% RSLogix 500 project CROWN_CITRUS_BIN_WASH_FROM_USB_AUG_30_2021_BAK438.RSS, saved by version 11.00.00.00 %
PROJECT "JBT BIN"    % processor: MicroLogix 1400 %

PROGRAM FILES
  LAD 2 "MAIN"  9 rungs
  LAD 3 "START_UP"  4 rungs
  LAD 4 "ENCODER"  6 rungs
  LAD 5 "CRADLE"  25 rungs
  LAD 6 "BRUSH"  7 rungs
  LAD 7 "TANK"  18 rungs
  LAD 8 "AUXILARY"  4 rungs
  LAD 9 "FAULTS"  29 rungs
  LAD 10 "HSC"  2 rungs

DATA FILES
  O0 OUTPUT  6 elements
  I1 INPUT  8 elements
  S2 STATUS  66 elements
  B3 BINARY  4 elements
  T4 TIMER  19 elements
  C5 COUNTER  1 elements
  R6 CONTROL  1 elements
  N7 INTEGER  7 elements
  F8 FLOAT  1 elements
  L9   3 elements
  L10   2 elements

LADDER 2 "MAIN"
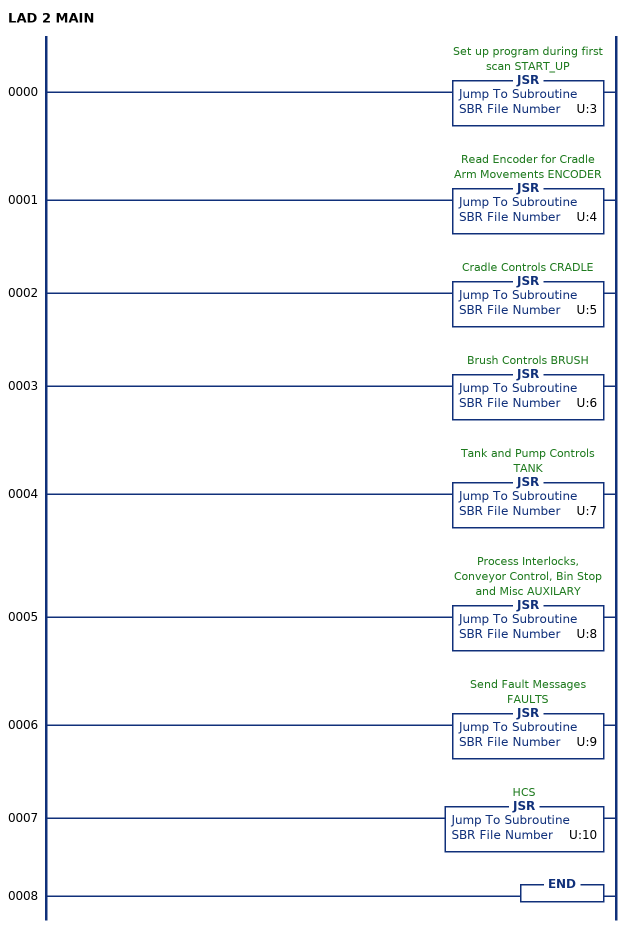
% Rung: 0 %
SOR JSR U:3 EOR
%   U:3  START_UP  "Set up program during first scan" %
% Rung: 1 %
SOR JSR U:4 EOR
%   U:4  ENCODER  "Read Encoder for Cradle Arm Movements" %
% Rung: 2 %
SOR JSR U:5 EOR
%   U:5  CRADLE  "Cradle Controls" %
% Rung: 3 %
SOR JSR U:6 EOR
%   U:6  BRUSH  "Brush Controls" %
% Rung: 4 %
SOR JSR U:7 EOR
%   U:7  TANK  "Tank and Pump Controls" %
% Rung: 5 %
SOR JSR U:8 EOR
%   U:8  AUXILARY  "Process Interlocks, Conveyor Control, Bin Stop and Misc" %
% Rung: 6 %
SOR JSR U:9 EOR
%   U:9  FAULTS  "Send Fault Messages" %
% Rung: 7 %
SOR JSR U:10 EOR
%   U:10  HCS %
% Rung: 8 %
SOR END EOR

LADDER 3 "START_UP"
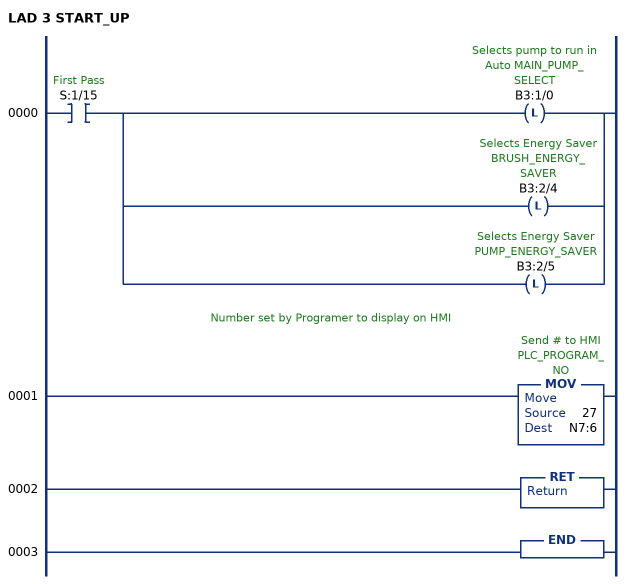
% Rung: 0 %
SOR XIC S:1/15 BST OTL B3:1/0 NXB BST OTL B3:2/4 NXB OTL B3:2/5 BND BND EOR
%   S:1/15  "First Pass" %
%   B3:1/0  MAIN_PUMP_SELECT  "Selects pump to run in Auto" %
%   B3:2/4  BRUSH_ENERGY_SAVER  "Selects Energy Saver" %
%   B3:2/5  PUMP_ENERGY_SAVER  "Selects Energy Saver" %
% Rung: 1 %
% Number set by Programer to display on HMI %
SOR MOV 27 N7:6 EOR
%   N7:6  PLC_PROGRAM_NO  "Send # to HMI" %
% Rung: 2 %
SOR RET EOR
% Rung: 3 %
SOR END EOR

LADDER 4 "ENCODER"
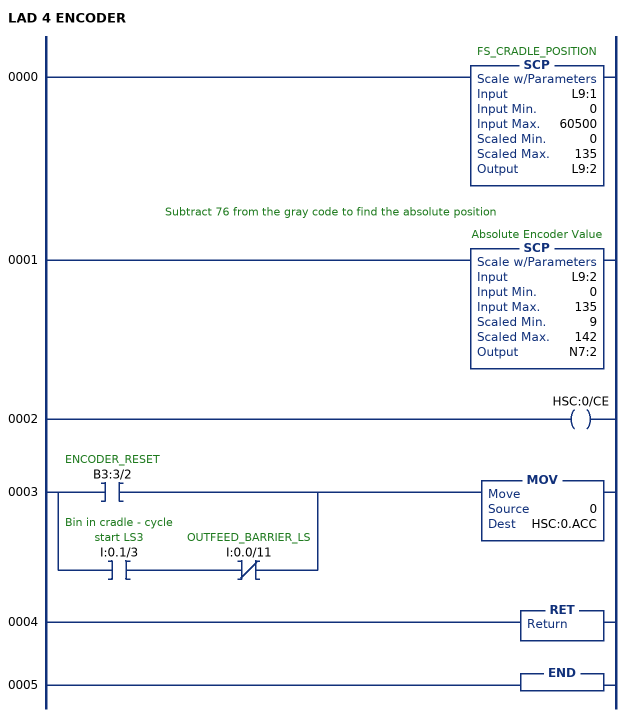
% Rung: 0 %
SOR SCP L9:1 0 60500 0 135 L9:2 EOR
%   L9:1  HSC_RAW_ACC %
%   L9:2  FS_CRADLE_POSITION %
% Rung: 1 %
% Subtract 76 from the gray code to find the absolute position %
SOR SCP L9:2 0 135 9 142 N7:2 EOR
%   L9:2  FS_CRADLE_POSITION %
%   N7:2  "Absolute Encoder Value" %
% Rung: 2 %
SOR OTE HSC:0/CE EOR
% Rung: 3 %
SOR BST XIC B3:3/2 NXB XIC I:0.1/3 XIO I:0.0/11 BND MOV 0 HSC:0.ACC EOR
%   B3:3/2  ENCODER_RESET %
%   I:0.1/3  LS3  "Bin in cradle - cycle start" %
%   I:0.0/11  OUTFEED_BARRIER_LS %
% Rung: 4 %
SOR RET EOR
% Rung: 5 %
SOR END EOR

LADDER 5 "CRADLE"
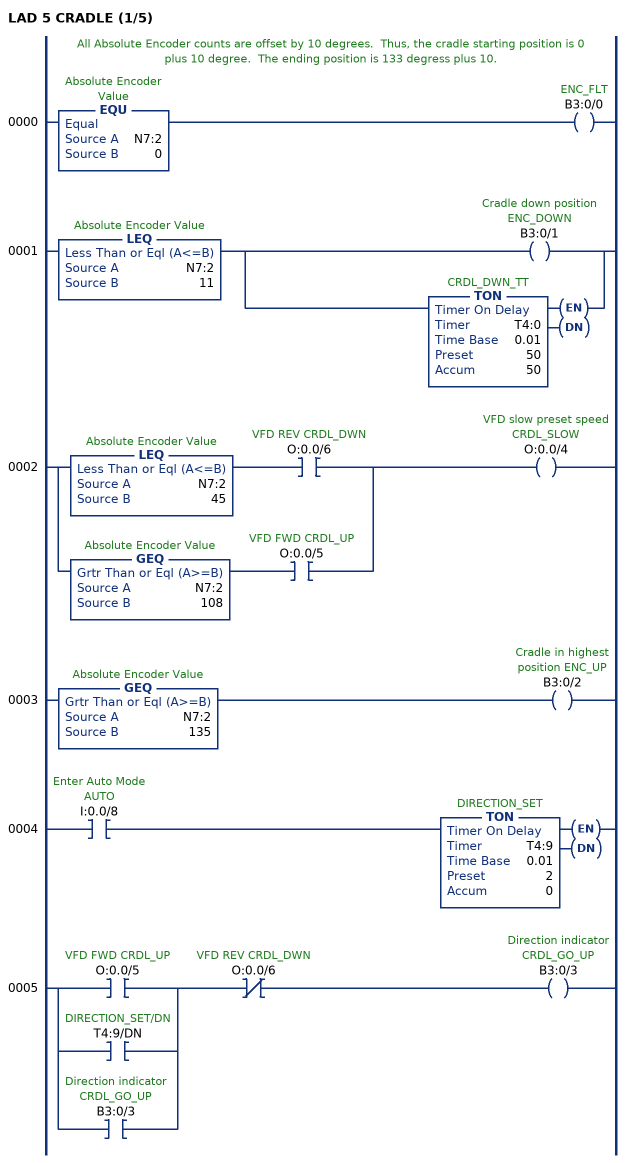
% Rung: 0 %
% All Absolute Encoder counts are offset by 10 degrees.  Thus, the cradle starting position is 0 plus 10 degree.  The ending position is 133 degress plus 10. %
SOR EQU N7:2 0 OTE B3:0/0 EOR
%   N7:2  "Absolute Encoder Value" %
%   B3:0/0  ENC_FLT %
% Rung: 1 %
SOR LEQ N7:2 11 BST OTE B3:0/1 NXB TON T4:0 0.01 50 50 BND EOR
%   N7:2  "Absolute Encoder Value" %
%   B3:0/1  ENC_DOWN  "Cradle down position" %
%   T4:0  CRDL_DWN_TT %
% Rung: 2 %
SOR BST LEQ N7:2 45 XIC O:0.0/6 NXB GEQ N7:2 108 XIC O:0.0/5 BND OTE O:0.0/4 EOR
%   N7:2  "Absolute Encoder Value" %
%   O:0.0/6  CRDL_DWN  "VFD REV" %
%   O:0.0/5  CRDL_UP  "VFD FWD" %
%   O:0.0/4  CRDL_SLOW  "VFD slow preset speed" %
% Rung: 3 %
SOR GEQ N7:2 135 OTE B3:0/2 EOR
%   N7:2  "Absolute Encoder Value" %
%   B3:0/2  ENC_UP  "Cradle in highest position" %
% Rung: 4 %
SOR XIC I:0.0/8 TON T4:9 0.01 2 0 EOR
%   I:0.0/8  AUTO  "Enter Auto Mode" %
%   T4:9  DIRECTION_SET %
% Rung: 5 %
SOR BST XIC O:0.0/5 NXB XIC T4:9/DN NXB XIC B3:0/3 BND XIO O:0.0/6 OTE B3:0/3 EOR
%   O:0.0/5  CRDL_UP  "VFD FWD" %
%   T4:9  DIRECTION_SET %
%   B3:0/3  CRDL_GO_UP  "Direction indicator" %
%   O:0.0/6  CRDL_DWN  "VFD REV" %

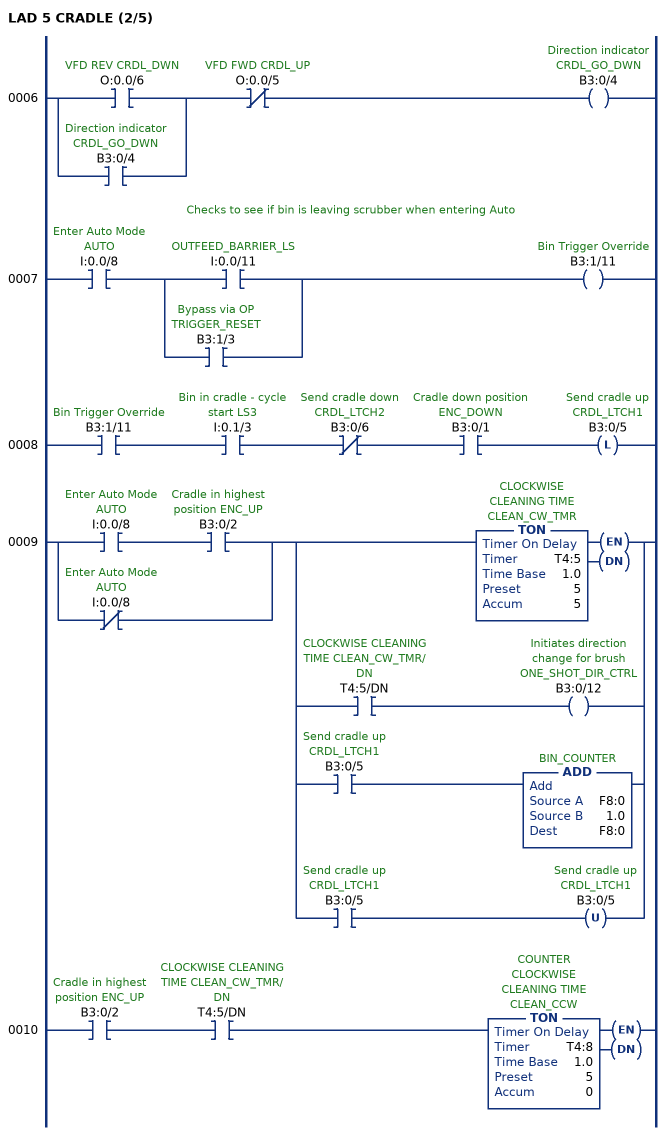
% Rung: 6 %
SOR BST XIC O:0.0/6 NXB XIC B3:0/4 BND XIO O:0.0/5 OTE B3:0/4 EOR
%   O:0.0/6  CRDL_DWN  "VFD REV" %
%   B3:0/4  CRDL_GO_DWN  "Direction indicator" %
%   O:0.0/5  CRDL_UP  "VFD FWD" %
% Rung: 7 %
% Checks to see if bin is leaving scrubber when entering Auto %
SOR XIC I:0.0/8 BST XIC I:0.0/11 NXB XIC B3:1/3 BND OTE B3:1/11 EOR
%   I:0.0/8  AUTO  "Enter Auto Mode" %
%   I:0.0/11  OUTFEED_BARRIER_LS %
%   B3:1/3  TRIGGER_RESET  "Bypass via OP" %
%   B3:1/11  "Bin Trigger Override" %
% Rung: 8 %
SOR XIC B3:1/11 XIC I:0.1/3 XIO B3:0/6 XIC B3:0/1 OTL B3:0/5 EOR
%   B3:1/11  "Bin Trigger Override" %
%   I:0.1/3  LS3  "Bin in cradle - cycle start" %
%   B3:0/6  CRDL_LTCH2  "Send cradle down" %
%   B3:0/1  ENC_DOWN  "Cradle down position" %
%   B3:0/5  CRDL_LTCH1  "Send cradle up" %
% Rung: 9 %
SOR BST XIC I:0.0/8 XIC B3:0/2 NXB XIO I:0.0/8 BND BST TON T4:5 1.0 5 5 NXB XIC T4:5/DN OTE B3:0/12 NXB BST XIC B3:0/5 ADD F8:0 1.0 F8:0 NXB XIC B3:0/5 OTU B3:0/5 BND BND EOR
%   I:0.0/8  AUTO  "Enter Auto Mode" %
%   B3:0/2  ENC_UP  "Cradle in highest position" %
%   T4:5  CLEAN_CW_TMR  "CLOCKWISE CLEANING TIME" %
%   B3:0/12  ONE_SHOT_DIR_CTRL  "Initiates direction change for brush" %
%   B3:0/5  CRDL_LTCH1  "Send cradle up" %
%   F8:0  BIN_COUNTER %
% Rung: 10 %
SOR XIC B3:0/2 XIC T4:5/DN TON T4:8 1.0 5 0 EOR
%   B3:0/2  ENC_UP  "Cradle in highest position" %
%   T4:5  CLEAN_CW_TMR  "CLOCKWISE CLEANING TIME" %
%   T4:8  CLEAN_CCW  "COUNTER CLOCKWISE CLEANING TIME" %

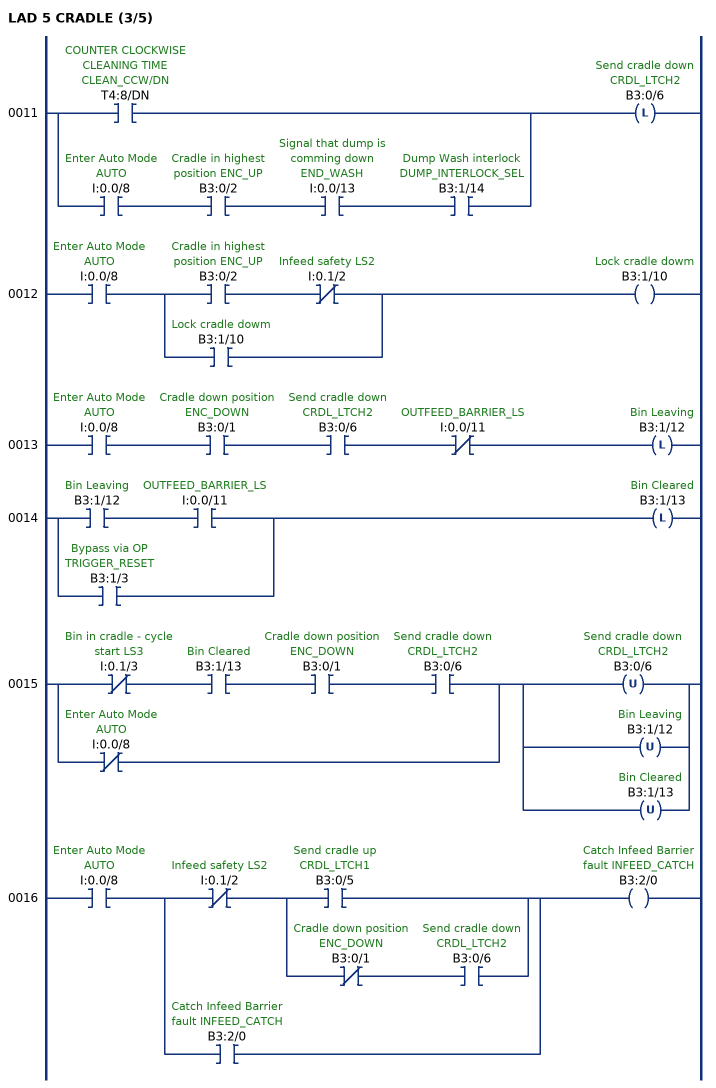
% Rung: 11 %
SOR BST XIC T4:8/DN NXB XIC I:0.0/8 XIC B3:0/2 XIC I:0.0/13 XIC B3:1/14 BND OTL B3:0/6 EOR
%   T4:8  CLEAN_CCW  "COUNTER CLOCKWISE CLEANING TIME" %
%   I:0.0/8  AUTO  "Enter Auto Mode" %
%   B3:0/2  ENC_UP  "Cradle in highest position" %
%   I:0.0/13  END_WASH  "Signal that dump is comming down" %
%   B3:1/14  DUMP_INTERLOCK_SEL  "Dump Wash interlock" %
%   B3:0/6  CRDL_LTCH2  "Send cradle down" %
% Rung: 12 %
SOR XIC I:0.0/8 BST XIC B3:0/2 XIO I:0.1/2 NXB XIC B3:1/10 BND OTE B3:1/10 EOR
%   I:0.0/8  AUTO  "Enter Auto Mode" %
%   B3:0/2  ENC_UP  "Cradle in highest position" %
%   I:0.1/2  LS2  "Infeed safety" %
%   B3:1/10  "Lock cradle dowm" %
% Rung: 13 %
SOR XIC I:0.0/8 XIC B3:0/1 XIC B3:0/6 XIO I:0.0/11 OTL B3:1/12 EOR
%   I:0.0/8  AUTO  "Enter Auto Mode" %
%   B3:0/1  ENC_DOWN  "Cradle down position" %
%   B3:0/6  CRDL_LTCH2  "Send cradle down" %
%   I:0.0/11  OUTFEED_BARRIER_LS %
%   B3:1/12  "Bin Leaving" %
% Rung: 14 %
SOR BST XIC B3:1/12 XIC I:0.0/11 NXB XIC B3:1/3 BND OTL B3:1/13 EOR
%   B3:1/12  "Bin Leaving" %
%   I:0.0/11  OUTFEED_BARRIER_LS %
%   B3:1/3  TRIGGER_RESET  "Bypass via OP" %
%   B3:1/13  "Bin Cleared" %
% Rung: 15 %
SOR BST XIO I:0.1/3 XIC B3:1/13 XIC B3:0/1 XIC B3:0/6 NXB XIO I:0.0/8 BND BST OTU B3:0/6 NXB BST OTU B3:1/12 NXB OTU B3:1/13 BND BND EOR
%   I:0.1/3  LS3  "Bin in cradle - cycle start" %
%   B3:1/13  "Bin Cleared" %
%   B3:0/1  ENC_DOWN  "Cradle down position" %
%   B3:0/6  CRDL_LTCH2  "Send cradle down" %
%   I:0.0/8  AUTO  "Enter Auto Mode" %
%   B3:1/12  "Bin Leaving" %
% Rung: 16 %
SOR XIC I:0.0/8 BST XIO I:0.1/2 BST XIC B3:0/5 NXB XIO B3:0/1 XIC B3:0/6 BND NXB XIC B3:2/0 BND OTE B3:2/0 EOR
%   I:0.0/8  AUTO  "Enter Auto Mode" %
%   I:0.1/2  LS2  "Infeed safety" %
%   B3:0/5  CRDL_LTCH1  "Send cradle up" %
%   B3:0/1  ENC_DOWN  "Cradle down position" %
%   B3:0/6  CRDL_LTCH2  "Send cradle down" %
%   B3:2/0  INFEED_CATCH  "Catch Infeed Barrier fault" %

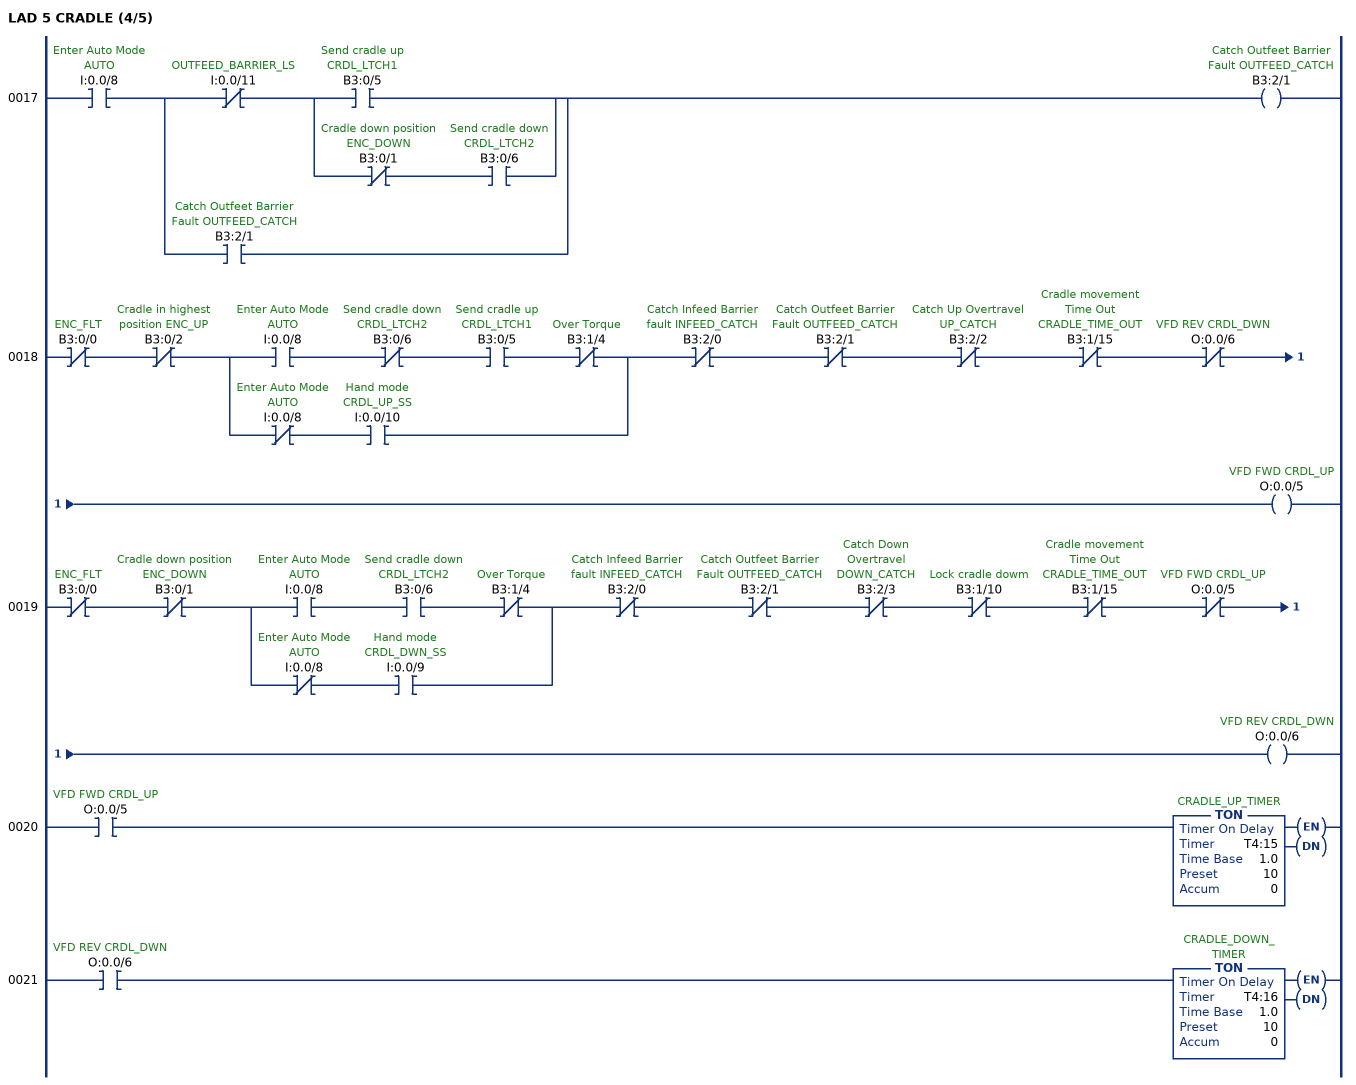
% Rung: 17 %
SOR XIC I:0.0/8 BST XIO I:0.0/11 BST XIC B3:0/5 NXB XIO B3:0/1 XIC B3:0/6 BND NXB XIC B3:2/1 BND OTE B3:2/1 EOR
%   I:0.0/8  AUTO  "Enter Auto Mode" %
%   I:0.0/11  OUTFEED_BARRIER_LS %
%   B3:0/5  CRDL_LTCH1  "Send cradle up" %
%   B3:0/1  ENC_DOWN  "Cradle down position" %
%   B3:0/6  CRDL_LTCH2  "Send cradle down" %
%   B3:2/1  OUTFEED_CATCH  "Catch Outfeet Barrier Fault" %
% Rung: 18 %
SOR XIO B3:0/0 XIO B3:0/2 BST XIC I:0.0/8 XIO B3:0/6 XIC B3:0/5 XIO B3:1/4 NXB XIO I:0.0/8 XIC I:0.0/10 BND XIO B3:2/0 XIO B3:2/1 XIO B3:2/2 XIO B3:1/15 XIO O:0.0/6 OTE O:0.0/5 EOR
%   B3:0/0  ENC_FLT %
%   B3:0/2  ENC_UP  "Cradle in highest position" %
%   I:0.0/8  AUTO  "Enter Auto Mode" %
%   B3:0/6  CRDL_LTCH2  "Send cradle down" %
%   B3:0/5  CRDL_LTCH1  "Send cradle up" %
%   B3:1/4  "Over Torque" %
%   I:0.0/10  CRDL_UP_SS  "Hand mode" %
%   B3:2/0  INFEED_CATCH  "Catch Infeed Barrier fault" %
%   B3:2/1  OUTFEED_CATCH  "Catch Outfeet Barrier Fault" %
%   B3:2/2  UP_CATCH  "Catch Up Overtravel" %
%   B3:1/15  CRADLE_TIME_OUT  "Cradle movement Time Out" %
%   O:0.0/6  CRDL_DWN  "VFD REV" %
%   O:0.0/5  CRDL_UP  "VFD FWD" %
% Rung: 19 %
SOR XIO B3:0/0 XIO B3:0/1 BST XIC I:0.0/8 XIC B3:0/6 XIO B3:1/4 NXB XIO I:0.0/8 XIC I:0.0/9 BND XIO B3:2/0 XIO B3:2/1 XIO B3:2/3 XIO B3:1/10 XIO B3:1/15 XIO O:0.0/5 OTE O:0.0/6 EOR
%   B3:0/0  ENC_FLT %
%   B3:0/1  ENC_DOWN  "Cradle down position" %
%   I:0.0/8  AUTO  "Enter Auto Mode" %
%   B3:0/6  CRDL_LTCH2  "Send cradle down" %
%   B3:1/4  "Over Torque" %
%   I:0.0/9  CRDL_DWN_SS  "Hand mode" %
%   B3:2/0  INFEED_CATCH  "Catch Infeed Barrier fault" %
%   B3:2/1  OUTFEED_CATCH  "Catch Outfeet Barrier Fault" %
%   B3:2/3  DOWN_CATCH  "Catch Down Overtravel" %
%   B3:1/10  "Lock cradle dowm" %
%   B3:1/15  CRADLE_TIME_OUT  "Cradle movement Time Out" %
%   O:0.0/5  CRDL_UP  "VFD FWD" %
%   O:0.0/6  CRDL_DWN  "VFD REV" %
% Rung: 20 %
SOR XIC O:0.0/5 TON T4:15 1.0 10 0 EOR
%   O:0.0/5  CRDL_UP  "VFD FWD" %
%   T4:15  CRADLE_UP_TIMER %
% Rung: 21 %
SOR XIC O:0.0/6 TON T4:16 1.0 10 0 EOR
%   O:0.0/6  CRDL_DWN  "VFD REV" %
%   T4:16  CRADLE_DOWN_TIMER %

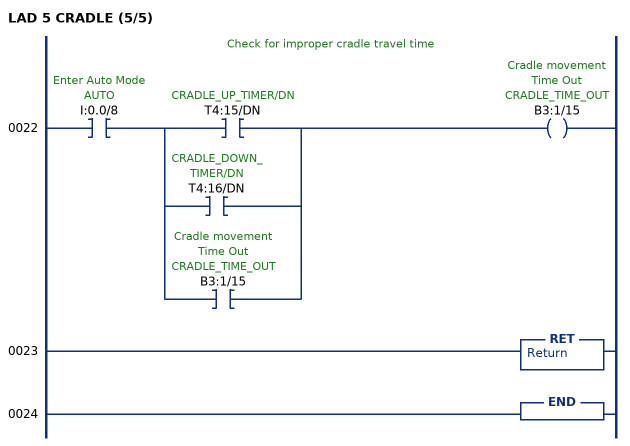
% Rung: 22 %
% Check for improper cradle travel time %
SOR XIC I:0.0/8 BST BST XIC T4:15/DN NXB XIC T4:16/DN BND NXB XIC B3:1/15 BND OTE B3:1/15 EOR
%   I:0.0/8  AUTO  "Enter Auto Mode" %
%   T4:15  CRADLE_UP_TIMER %
%   T4:16  CRADLE_DOWN_TIMER %
%   B3:1/15  CRADLE_TIME_OUT  "Cradle movement Time Out" %
% Rung: 23 %
SOR RET EOR
% Rung: 24 %
SOR END EOR

LADDER 6 "BRUSH"
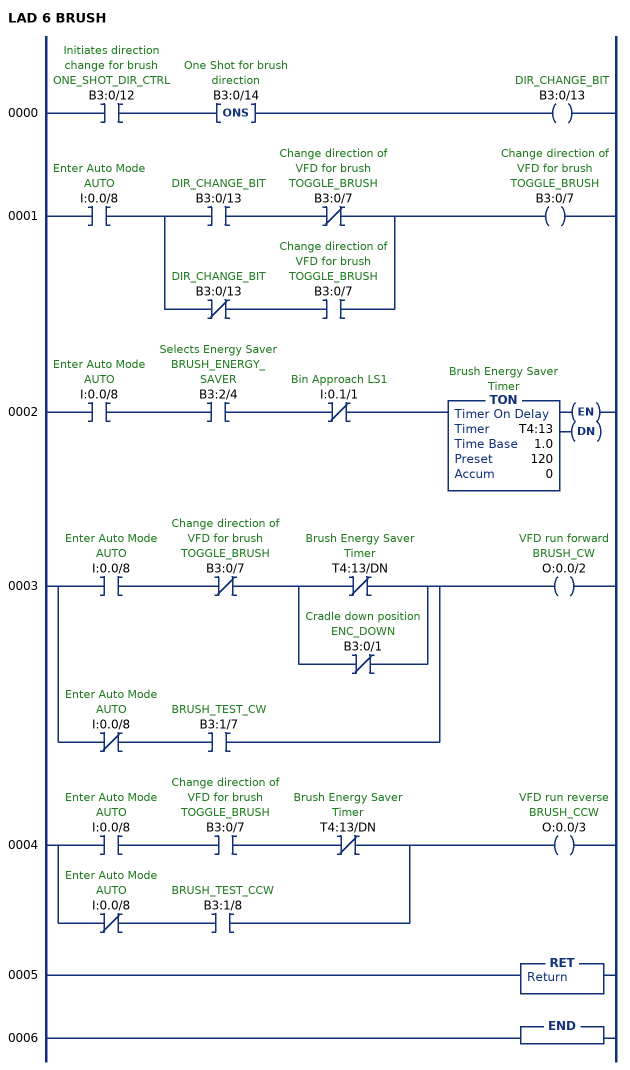
% Rung: 0 %
SOR XIC B3:0/12 ONS B3:0/14 OTE B3:0/13 EOR
%   B3:0/12  ONE_SHOT_DIR_CTRL  "Initiates direction change for brush" %
%   B3:0/14  "One Shot for brush direction" %
%   B3:0/13  DIR_CHANGE_BIT %
% Rung: 1 %
SOR XIC I:0.0/8 BST XIC B3:0/13 XIO B3:0/7 NXB XIO B3:0/13 XIC B3:0/7 BND OTE B3:0/7 EOR
%   I:0.0/8  AUTO  "Enter Auto Mode" %
%   B3:0/13  DIR_CHANGE_BIT %
%   B3:0/7  TOGGLE_BRUSH  "Change direction of VFD for brush" %
% Rung: 2 %
SOR XIC I:0.0/8 XIC B3:2/4 XIO I:0.1/1 TON T4:13 1.0 120 0 EOR
%   I:0.0/8  AUTO  "Enter Auto Mode" %
%   B3:2/4  BRUSH_ENERGY_SAVER  "Selects Energy Saver" %
%   I:0.1/1  LS1  "Bin Approach" %
%   T4:13  "Brush Energy Saver Timer" %
% Rung: 3 %
SOR BST XIC I:0.0/8 XIO B3:0/7 BST XIO T4:13/DN NXB XIO B3:0/1 BND NXB XIO I:0.0/8 XIC B3:1/7 BND OTE O:0.0/2 EOR
%   I:0.0/8  AUTO  "Enter Auto Mode" %
%   B3:0/7  TOGGLE_BRUSH  "Change direction of VFD for brush" %
%   T4:13  "Brush Energy Saver Timer" %
%   B3:0/1  ENC_DOWN  "Cradle down position" %
%   B3:1/7  BRUSH_TEST_CW %
%   O:0.0/2  BRUSH_CW  "VFD run forward" %
% Rung: 4 %
SOR BST XIC I:0.0/8 XIC B3:0/7 XIO T4:13/DN NXB XIO I:0.0/8 XIC B3:1/8 BND OTE O:0.0/3 EOR
%   I:0.0/8  AUTO  "Enter Auto Mode" %
%   B3:0/7  TOGGLE_BRUSH  "Change direction of VFD for brush" %
%   T4:13  "Brush Energy Saver Timer" %
%   B3:1/8  BRUSH_TEST_CCW %
%   O:0.0/3  BRUSH_CCW  "VFD run reverse" %
% Rung: 5 %
SOR RET EOR
% Rung: 6 %
SOR END EOR

LADDER 7 "TANK"
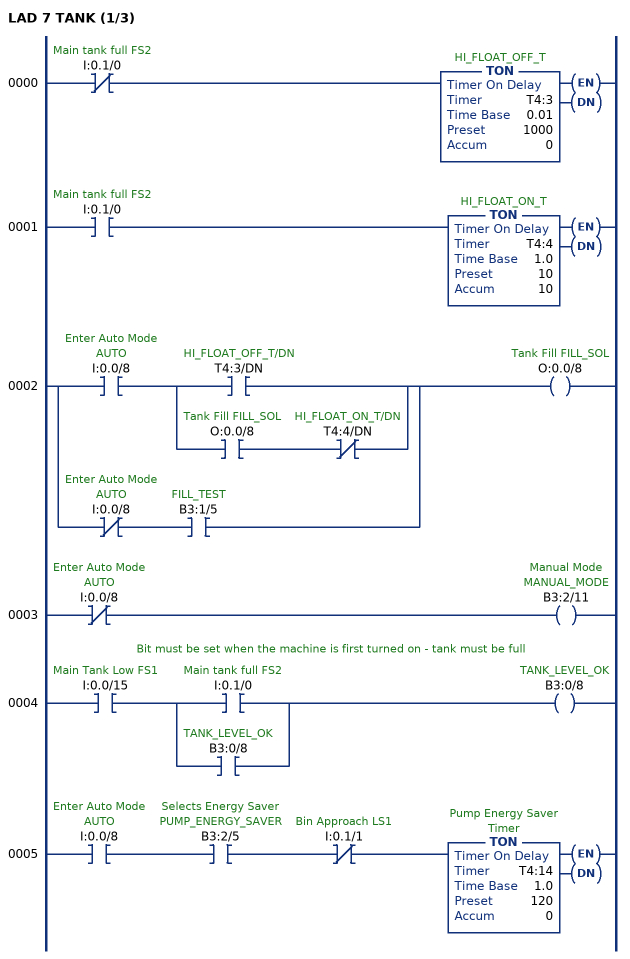
% Rung: 0 %
SOR XIO I:0.1/0 TON T4:3 0.01 1000 0 EOR
%   I:0.1/0  FS2  "Main tank full" %
%   T4:3  HI_FLOAT_OFF_T %
% Rung: 1 %
SOR XIC I:0.1/0 TON T4:4 1.0 10 10 EOR
%   I:0.1/0  FS2  "Main tank full" %
%   T4:4  HI_FLOAT_ON_T %
% Rung: 2 %
SOR BST XIC I:0.0/8 BST XIC T4:3/DN NXB XIC O:0.0/8 XIO T4:4/DN BND NXB XIO I:0.0/8 XIC B3:1/5 BND OTE O:0.0/8 EOR
%   I:0.0/8  AUTO  "Enter Auto Mode" %
%   T4:3  HI_FLOAT_OFF_T %
%   O:0.0/8  FILL_SOL  "Tank Fill" %
%   T4:4  HI_FLOAT_ON_T %
%   B3:1/5  FILL_TEST %
% Rung: 3 %
SOR XIO I:0.0/8 OTE B3:2/11 EOR
%   I:0.0/8  AUTO  "Enter Auto Mode" %
%   B3:2/11  MANUAL_MODE  "Manual Mode" %
% Rung: 4 %
% Bit must be set when the machine is first turned on - tank must be full %
SOR XIC I:0.0/15 BST XIC I:0.1/0 NXB XIC B3:0/8 BND OTE B3:0/8 EOR
%   I:0.0/15  FS1  "Main Tank Low" %
%   I:0.1/0  FS2  "Main tank full" %
%   B3:0/8  TANK_LEVEL_OK %
% Rung: 5 %
SOR XIC I:0.0/8 XIC B3:2/5 XIO I:0.1/1 TON T4:14 1.0 120 0 EOR
%   I:0.0/8  AUTO  "Enter Auto Mode" %
%   B3:2/5  PUMP_ENERGY_SAVER  "Selects Energy Saver" %
%   I:0.1/1  LS1  "Bin Approach" %
%   T4:14  "Pump Energy Saver Timer" %

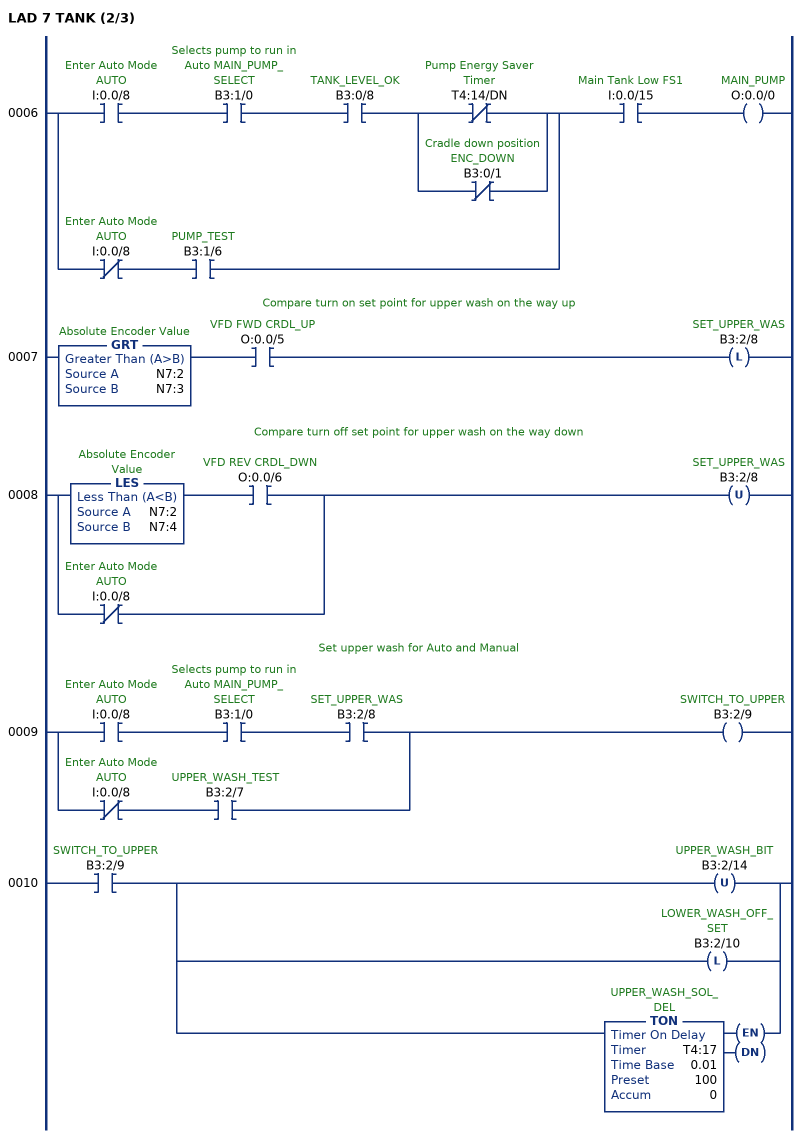
% Rung: 6 %
SOR BST XIC I:0.0/8 XIC B3:1/0 XIC B3:0/8 BST XIO T4:14/DN NXB XIO B3:0/1 BND NXB XIO I:0.0/8 XIC B3:1/6 BND XIC I:0.0/15 OTE O:0.0/0 EOR
%   I:0.0/8  AUTO  "Enter Auto Mode" %
%   B3:1/0  MAIN_PUMP_SELECT  "Selects pump to run in Auto" %
%   B3:0/8  TANK_LEVEL_OK %
%   T4:14  "Pump Energy Saver Timer" %
%   B3:0/1  ENC_DOWN  "Cradle down position" %
%   B3:1/6  PUMP_TEST %
%   I:0.0/15  FS1  "Main Tank Low" %
%   O:0.0/0  MAIN_PUMP %
% Rung: 7 %
% Compare turn on set point for upper wash on the way up %
SOR GRT N7:2 N7:3 XIC O:0.0/5 OTL B3:2/8 EOR
%   N7:2  "Absolute Encoder Value" %
%   N7:3  UPPER_WASH_TURN_ON %
%   O:0.0/5  CRDL_UP  "VFD FWD" %
%   B3:2/8  SET_UPPER_WAS %
% Rung: 8 %
% Compare turn off set point for upper wash on the way down %
SOR BST LES N7:2 N7:4 XIC O:0.0/6 NXB XIO I:0.0/8 BND OTU B3:2/8 EOR
%   N7:2  "Absolute Encoder Value" %
%   N7:4  UPPER_WASH_TURN_OFF %
%   O:0.0/6  CRDL_DWN  "VFD REV" %
%   I:0.0/8  AUTO  "Enter Auto Mode" %
%   B3:2/8  SET_UPPER_WAS %
% Rung: 9 %
% Set upper wash for Auto and Manual %
SOR BST XIC I:0.0/8 XIC B3:1/0 XIC B3:2/8 NXB XIO I:0.0/8 XIC B3:2/7 BND OTE B3:2/9 EOR
%   I:0.0/8  AUTO  "Enter Auto Mode" %
%   B3:1/0  MAIN_PUMP_SELECT  "Selects pump to run in Auto" %
%   B3:2/8  SET_UPPER_WAS %
%   B3:2/7  UPPER_WASH_TEST %
%   B3:2/9  SWITCH_TO_UPPER %
% Rung: 10 %
SOR XIC B3:2/9 BST OTU B3:2/14 NXB BST OTL B3:2/10 NXB TON T4:17 0.01 100 0 BND BND EOR
%   B3:2/9  SWITCH_TO_UPPER %
%   B3:2/14  UPPER_WASH_BIT %
%   B3:2/10  LOWER_WASH_OFF_SET %
%   T4:17  UPPER_WASH_SOL_DEL %

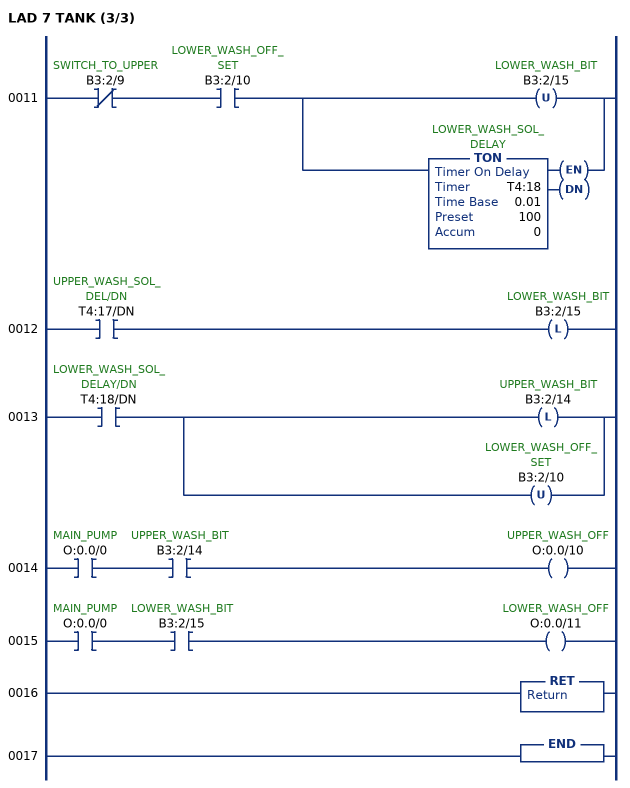
% Rung: 11 %
SOR XIO B3:2/9 XIC B3:2/10 BST OTU B3:2/15 NXB TON T4:18 0.01 100 0 BND EOR
%   B3:2/9  SWITCH_TO_UPPER %
%   B3:2/10  LOWER_WASH_OFF_SET %
%   B3:2/15  LOWER_WASH_BIT %
%   T4:18  LOWER_WASH_SOL_DELAY %
% Rung: 12 %
SOR XIC T4:17/DN OTL B3:2/15 EOR
%   T4:17  UPPER_WASH_SOL_DEL %
%   B3:2/15  LOWER_WASH_BIT %
% Rung: 13 %
SOR XIC T4:18/DN BST OTL B3:2/14 NXB OTU B3:2/10 BND EOR
%   T4:18  LOWER_WASH_SOL_DELAY %
%   B3:2/14  UPPER_WASH_BIT %
%   B3:2/10  LOWER_WASH_OFF_SET %
% Rung: 14 %
SOR XIC O:0.0/0 XIC B3:2/14 OTE O:0.0/10 EOR
%   O:0.0/0  MAIN_PUMP %
%   B3:2/14  UPPER_WASH_BIT %
%   O:0.0/10  UPPER_WASH_OFF %
% Rung: 15 %
SOR XIC O:0.0/0 XIC B3:2/15 OTE O:0.0/11 EOR
%   O:0.0/0  MAIN_PUMP %
%   B3:2/15  LOWER_WASH_BIT %
%   O:0.0/11  LOWER_WASH_OFF %
% Rung: 16 %
SOR RET EOR
% Rung: 17 %
SOR END EOR

LADDER 8 "AUXILARY"
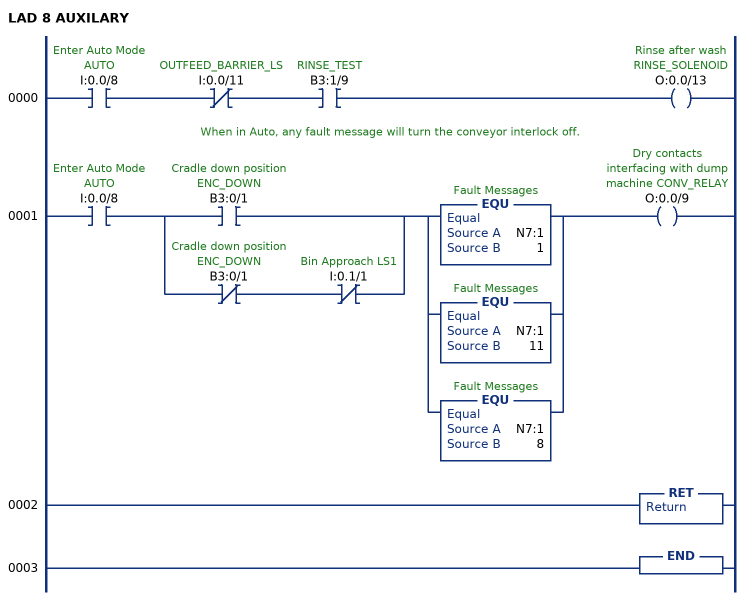
% Rung: 0 %
SOR XIC I:0.0/8 XIO I:0.0/11 XIC B3:1/9 OTE O:0.0/13 EOR
%   I:0.0/8  AUTO  "Enter Auto Mode" %
%   I:0.0/11  OUTFEED_BARRIER_LS %
%   B3:1/9  RINSE_TEST %
%   O:0.0/13  RINSE_SOLENOID  "Rinse after wash" %
% Rung: 1 %
% When in Auto, any fault message will turn the conveyor interlock off. %
SOR XIC I:0.0/8 BST XIC B3:0/1 NXB XIO B3:0/1 XIO I:0.1/1 BND BST EQU N7:1 1 NXB BST EQU N7:1 11 NXB EQU N7:1 8 BND BND OTE O:0.0/9 EOR
%   I:0.0/8  AUTO  "Enter Auto Mode" %
%   B3:0/1  ENC_DOWN  "Cradle down position" %
%   I:0.1/1  LS1  "Bin Approach" %
%   N7:1  "Fault Messages" %
%   O:0.0/9  CONV_RELAY  "Dry contacts interfacing with dump machine" %
% Rung: 2 %
SOR RET EOR
% Rung: 3 %
SOR END EOR

LADDER 9 "FAULTS"
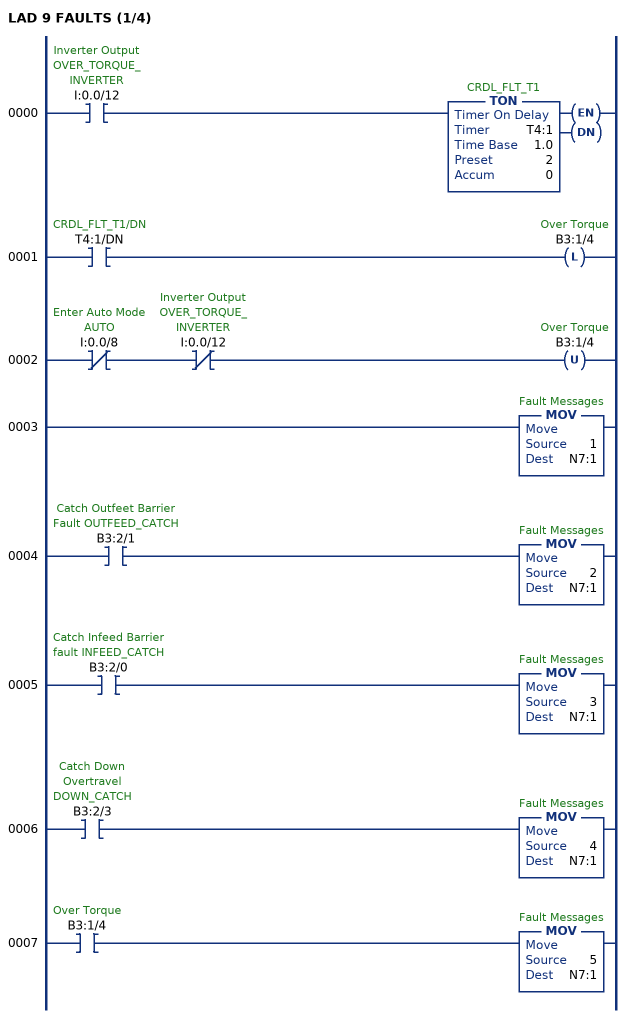
% Rung: 0 %
SOR XIC I:0.0/12 TON T4:1 1.0 2 0 EOR
%   I:0.0/12  OVER_TORQUE_INVERTER  "Inverter Output" %
%   T4:1  CRDL_FLT_T1 %
% Rung: 1 %
SOR XIC T4:1/DN OTL B3:1/4 EOR
%   T4:1  CRDL_FLT_T1 %
%   B3:1/4  "Over Torque" %
% Rung: 2 %
SOR XIO I:0.0/8 XIO I:0.0/12 OTU B3:1/4 EOR
%   I:0.0/8  AUTO  "Enter Auto Mode" %
%   I:0.0/12  OVER_TORQUE_INVERTER  "Inverter Output" %
%   B3:1/4  "Over Torque" %
% Rung: 3 %
SOR MOV 1 N7:1 EOR
%   N7:1  "Fault Messages" %
% Rung: 4 %
SOR XIC B3:2/1 MOV 2 N7:1 EOR
%   B3:2/1  OUTFEED_CATCH  "Catch Outfeet Barrier Fault" %
%   N7:1  "Fault Messages" %
% Rung: 5 %
SOR XIC B3:2/0 MOV 3 N7:1 EOR
%   B3:2/0  INFEED_CATCH  "Catch Infeed Barrier fault" %
%   N7:1  "Fault Messages" %
% Rung: 6 %
SOR XIC B3:2/3 MOV 4 N7:1 EOR
%   B3:2/3  DOWN_CATCH  "Catch Down Overtravel" %
%   N7:1  "Fault Messages" %
% Rung: 7 %
SOR XIC B3:1/4 MOV 5 N7:1 EOR
%   B3:1/4  "Over Torque" %
%   N7:1  "Fault Messages" %

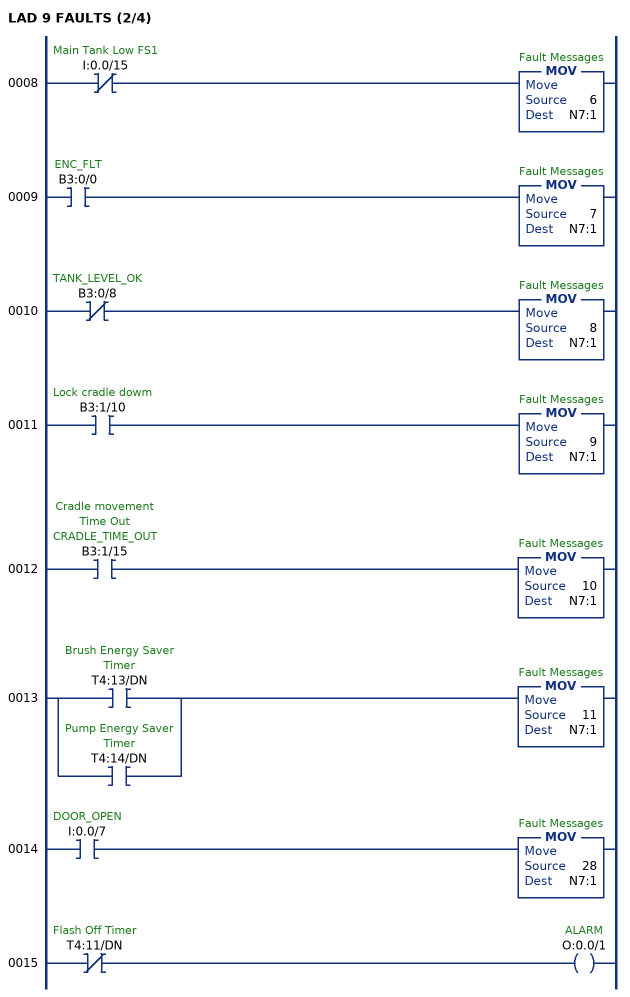
% Rung: 8 %
SOR XIO I:0.0/15 MOV 6 N7:1 EOR
%   I:0.0/15  FS1  "Main Tank Low" %
%   N7:1  "Fault Messages" %
% Rung: 9 %
SOR XIC B3:0/0 MOV 7 N7:1 EOR
%   B3:0/0  ENC_FLT %
%   N7:1  "Fault Messages" %
% Rung: 10 %
SOR XIO B3:0/8 MOV 8 N7:1 EOR
%   B3:0/8  TANK_LEVEL_OK %
%   N7:1  "Fault Messages" %
% Rung: 11 %
SOR XIC B3:1/10 MOV 9 N7:1 EOR
%   B3:1/10  "Lock cradle dowm" %
%   N7:1  "Fault Messages" %
% Rung: 12 %
SOR XIC B3:1/15 MOV 10 N7:1 EOR
%   B3:1/15  CRADLE_TIME_OUT  "Cradle movement Time Out" %
%   N7:1  "Fault Messages" %
% Rung: 13 %
SOR BST XIC T4:13/DN NXB XIC T4:14/DN BND MOV 11 N7:1 EOR
%   T4:13  "Brush Energy Saver Timer" %
%   T4:14  "Pump Energy Saver Timer" %
%   N7:1  "Fault Messages" %
% Rung: 14 %
SOR XIC I:0.0/7 MOV 28 N7:1 EOR
%   I:0.0/7  DOOR_OPEN %
%   N7:1  "Fault Messages" %
% Rung: 15 %
SOR XIO T4:11/DN OTE O:0.0/1 EOR
%   T4:11  "Flash Off Timer" %
%   O:0.0/1  ALARM %

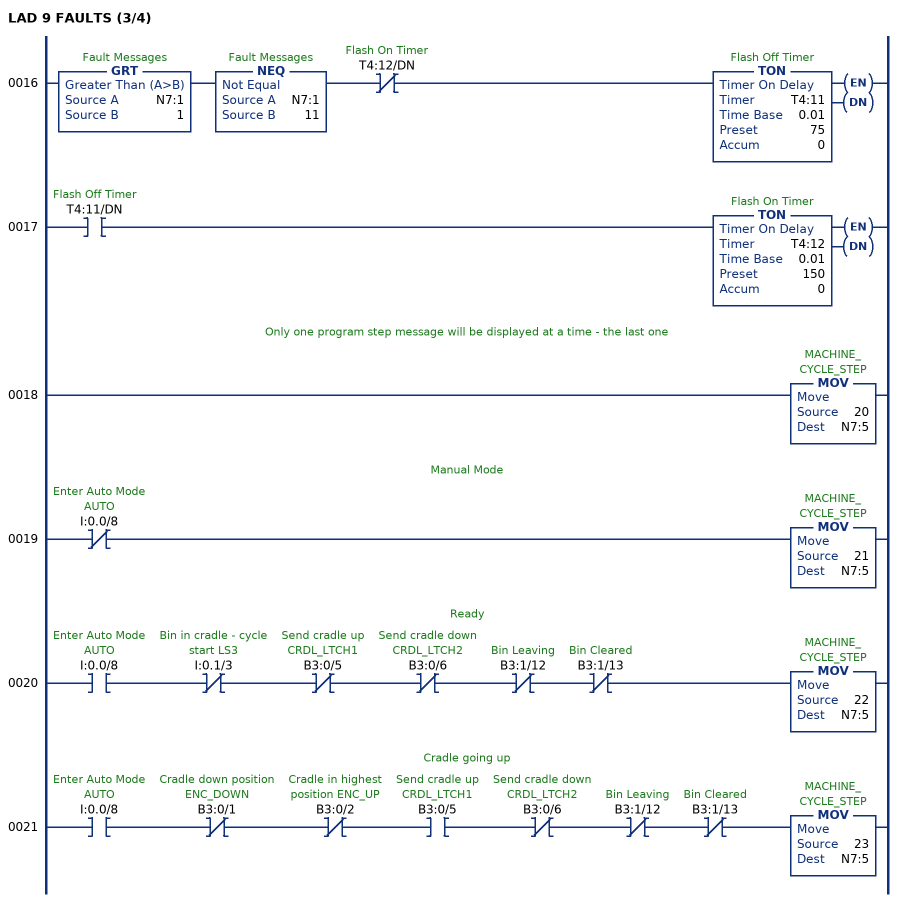
% Rung: 16 %
SOR GRT N7:1 1 NEQ N7:1 11 XIO T4:12/DN TON T4:11 0.01 75 0 EOR
%   N7:1  "Fault Messages" %
%   T4:12  "Flash On Timer" %
%   T4:11  "Flash Off Timer" %
% Rung: 17 %
SOR XIC T4:11/DN TON T4:12 0.01 150 0 EOR
%   T4:11  "Flash Off Timer" %
%   T4:12  "Flash On Timer" %
% Rung: 18 %
% Only one program step message will be displayed at a time - the last one %
SOR MOV 20 N7:5 EOR
%   N7:5  MACHINE_CYCLE_STEP %
% Rung: 19 %
% Manual Mode %
SOR XIO I:0.0/8 MOV 21 N7:5 EOR
%   I:0.0/8  AUTO  "Enter Auto Mode" %
%   N7:5  MACHINE_CYCLE_STEP %
% Rung: 20 %
% Ready %
SOR XIC I:0.0/8 XIO I:0.1/3 XIO B3:0/5 XIO B3:0/6 XIO B3:1/12 XIO B3:1/13 MOV 22 N7:5 EOR
%   I:0.0/8  AUTO  "Enter Auto Mode" %
%   I:0.1/3  LS3  "Bin in cradle - cycle start" %
%   B3:0/5  CRDL_LTCH1  "Send cradle up" %
%   B3:0/6  CRDL_LTCH2  "Send cradle down" %
%   B3:1/12  "Bin Leaving" %
%   B3:1/13  "Bin Cleared" %
%   N7:5  MACHINE_CYCLE_STEP %
% Rung: 21 %
% Cradle going up %
SOR XIC I:0.0/8 XIO B3:0/1 XIO B3:0/2 XIC B3:0/5 XIO B3:0/6 XIO B3:1/12 XIO B3:1/13 MOV 23 N7:5 EOR
%   I:0.0/8  AUTO  "Enter Auto Mode" %
%   B3:0/1  ENC_DOWN  "Cradle down position" %
%   B3:0/2  ENC_UP  "Cradle in highest position" %
%   B3:0/5  CRDL_LTCH1  "Send cradle up" %
%   B3:0/6  CRDL_LTCH2  "Send cradle down" %
%   B3:1/12  "Bin Leaving" %
%   B3:1/13  "Bin Cleared" %
%   N7:5  MACHINE_CYCLE_STEP %

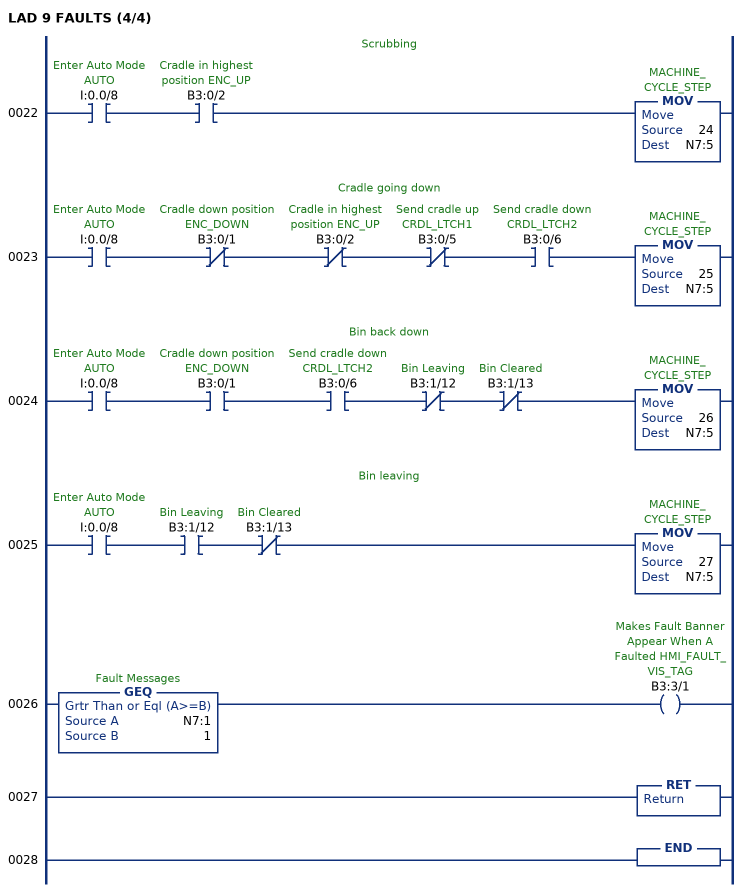
% Rung: 22 %
% Scrubbing %
SOR XIC I:0.0/8 XIC B3:0/2 MOV 24 N7:5 EOR
%   I:0.0/8  AUTO  "Enter Auto Mode" %
%   B3:0/2  ENC_UP  "Cradle in highest position" %
%   N7:5  MACHINE_CYCLE_STEP %
% Rung: 23 %
% Cradle going down %
SOR XIC I:0.0/8 XIO B3:0/1 XIO B3:0/2 XIO B3:0/5 XIC B3:0/6 MOV 25 N7:5 EOR
%   I:0.0/8  AUTO  "Enter Auto Mode" %
%   B3:0/1  ENC_DOWN  "Cradle down position" %
%   B3:0/2  ENC_UP  "Cradle in highest position" %
%   B3:0/5  CRDL_LTCH1  "Send cradle up" %
%   B3:0/6  CRDL_LTCH2  "Send cradle down" %
%   N7:5  MACHINE_CYCLE_STEP %
% Rung: 24 %
% Bin back down %
SOR XIC I:0.0/8 XIC B3:0/1 XIC B3:0/6 XIO B3:1/12 XIO B3:1/13 MOV 26 N7:5 EOR
%   I:0.0/8  AUTO  "Enter Auto Mode" %
%   B3:0/1  ENC_DOWN  "Cradle down position" %
%   B3:0/6  CRDL_LTCH2  "Send cradle down" %
%   B3:1/12  "Bin Leaving" %
%   B3:1/13  "Bin Cleared" %
%   N7:5  MACHINE_CYCLE_STEP %
% Rung: 25 %
% Bin leaving %
SOR XIC I:0.0/8 XIC B3:1/12 XIO B3:1/13 MOV 27 N7:5 EOR
%   I:0.0/8  AUTO  "Enter Auto Mode" %
%   B3:1/12  "Bin Leaving" %
%   B3:1/13  "Bin Cleared" %
%   N7:5  MACHINE_CYCLE_STEP %
% Rung: 26 %
SOR GEQ N7:1 1 OTE B3:3/1 EOR
%   N7:1  "Fault Messages" %
%   B3:3/1  HMI_FAULT_VIS_TAG  "Makes Fault Banner Appear When A Faulted" %
% Rung: 27 %
SOR RET EOR
% Rung: 28 %
SOR END EOR

LADDER 10 "HSC"
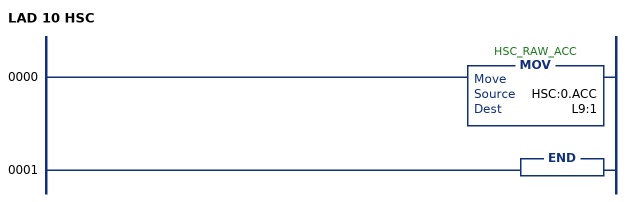
% Rung: 0 %
SOR MOV HSC:0.ACC L9:1 EOR
%   L9:1  HSC_RAW_ACC %
% Rung: 1 %
SOR END EOR

OTHER DOCUMENTED ADDRESSES
  B3:0/9  SANITIZE_LTCH  "Triggered by reset limit sw."
  B3:0/10  SANITIZE_BIT  "Allow crdl ltch2 to unlatch only once until sanitize cycle is over"
  B3:0/11  CRDL_EN  "mcr on and no encoder fault"
  B3:0/15  CRDL_HAND_SS
  B3:1/1  RINSE_SELECT  "Turn ON Rinse"
  B3:1/2  TRIGGER_OVERRIDE  "Bypass via OP"
  B3:3/0  OPEN_CONTACT  "Machine not Equipt with OT LS"
  C5:0/CU  EVENT_COUNTER
  I:0.0/0  ENC_BIT0
  I:0.0/1  ENC_BIT1
  I:0.0/5  HOME_SENSOR
  L10:1/1  FAULT_MESSAGES
  N7:0  ENC_POS
  N7:0/1  "DEC2"
  N7:0/2  "DEC4"
  N7:0/3  "DEC8"
  N7:0/4  "DEC16"
  N7:0/5  "DEC32"
  N7:0/6  "DEC64"
  N7:0/7  "DEC128"
  N7:1/0  "Fault-Infeed Blocked"
  N7:1/1  "Fault-Outfeed Blocked"
  N7:1/2  "Fault-Cradle Overtravel Up"
  N7:1/3  "Fault-Cradle Overtravel down"
  N7:1/4  "Fault-Torque Cradle Inverter"
  N7:1/5  "Main Tank Low"
  N7:1/6  "Encoder Fault"
  N7:1/7  "Fill Main Tank"
  N7:7  LOWER_WASH_TURN_OFF
  N9:0  K1
  O:0.0/7  NOT_USED
  T4:0/EN  CRDL_DWN_T  "Allows cradle to set down completely before conv starts"
  T4:2  CRDL_FLT_T2
  T4:6  SANITIZE_T
  T4:7  CRDL_DWN_T2  "Inhibits cradle up for 5 sec. after cradle sets down"
  T4:10  CRADLE_TIMER  "Cradle travel watch dog timer"

COMMENTS NOT ATTACHED TO A CURRENT RUNG
  T4:6.PRE: As long as the bit is set, the message will be displayed.  Bit #1 is Message #1.  Bit #3 is message #4.  Binary to decimal.
  N7:1/0: As long as the bit is set, the message will be displayed.  Bit #1 is Message #1.  Bit #3 is message #4.  Binary to decimal.
  T4:7: Timer not used
  N7:0/7: Read all 8 bits of the Encoder and convert to Gray Code

REVISION NOTES
  0: Added barrier and overtravel tatches
  1: Added indepentent barrier and overtravel catches
  2: Changed ffrom Panel #8.  Added B3:0/1 to prevent B3:0/5 from latching up while cradle is not down
  3: Added more troubleshooting help - step sequences
  4: Costa Rica Panel #19 with individual upper and lower wash solenoids

DATA TABLE (non-zero values as saved)
DATA B3
% B3:0 % 0X5D02 0X0203 0X4830 0X0002
DATA T4
% .PRE .ACC %
% T4:0 % 50 50
% T4:1 % 2 0
% T4:2 % 1 0
% T4:3 % 1000 0
% T4:4 % 10 10
% T4:5 % 5 5
% T4:6 % 658 0
% T4:7 % 375 500
% T4:8 % 5 0
% T4:9 % 2 0
% T4:10 % 500 0
% T4:11 % 75 0
% T4:12 % 150 0
% T4:13 % 120 0
% T4:14 % 120 0
% T4:15 % 10 0
% T4:16 % 10 0
% T4:17 % 100 0
% T4:18 % 100 0
DATA N7
% N7:0 % 219 1 9 65 130 21 27
DATA F8
% F8:0 % 34
